# B&R Automation Studio project plcProject
Automation Studio 4.9

## Configuration Simulator

### Task classes (Cpu.sw)
```
Cyclic#4:
  Logic <- Logic.prg
VcDataObjects: Hmi <- Hmi.dob
```

### Hardware
```
PC : PC_any v1.1.1.0 (OrderNumber=PC)
  Connector IF3:
    Vnc1
    VncVcObjectName1 = Hmi
    VncKeyMappingFile1 = VC\PS2-Keyboard.dis
    VncAuthentication1 = 1
    VncPasswordViewOnly1 = 0
    VncPasswordViewControl1 = 1
    VncRefreshRate1 = 100
  ConfigurationID = plcProject_Simulator
  FileDevice1
  FileDeviceName1 = USER
  FileDevicePath1 = USER_PATH
```

## Logical view

### Program Logical/Logic (IEC)

#### Variables.var
```iecst
VAR
	reset : BOOL;
	countUp : BOOL;
	counter : USINT;
END_VAR
```

#### Main.st
```iecst
PROGRAM _CYCLIC

	IF (countUp) THEN
		countUp := FALSE;
		counter := counter + 1;
	END_IF

	IF (reset) THEN
		reset := FALSE;
		counter := 0;
	END_IF

END_PROGRAM
```

- Visualisation Logical/Hmi (not shown)

Listed in the project but not available here: Logical/Global.typ, Logical/Global.var, Logical/Libraries
